(* CODESYS project T1_ARC.project

Project tree, tasks and I/O mapping:
  Device : CODESYS Control Win V3, 3S - Smart Software Solutions GmbH, order no. 305021, version 3.5.7.20
    application Application
      libraries: Standard, * (System); Util, * (System)
      task MainTask (cyclic, interval t#20ms, priority 1) calls PLC_PRG
      program PLC_PRG [FBD]
      global variables GVL_ARC
      Symbols
*)

// Device/Application/GVL_ARC
VAR_GLOBAL
	PV_h: REAL;
	SP_h: REAL;
	KP_h: REAL;
	TN_h: REAL;
	TV_h: REAL;
	u1_MAN: REAL;
	MAN: BOOL;
	RES: BOOL;
	u1_h: REAL;
	PV_K: REAL;
	SP_K: REAL;
	KP_K: REAL;
	TN_K: REAL;
	TV_K: REAL;
	K_MAN: REAL;
	K: REAL;
	PV_f2: REAL;
	SP_f2: REAL;
	KP_f2: REAL;
	TN_f2: REAL;
	TV_f2: REAL;
	f2_MAN: REAL;
	u2: REAL;
	PV_f1: REAL;
END_VAR

// Device/Application/PLC_PRG
PROGRAM PLC_PRG
VAR
	PID_h: PID;
	PID_K: PID;
	PID_f2: PID;
END_VAR

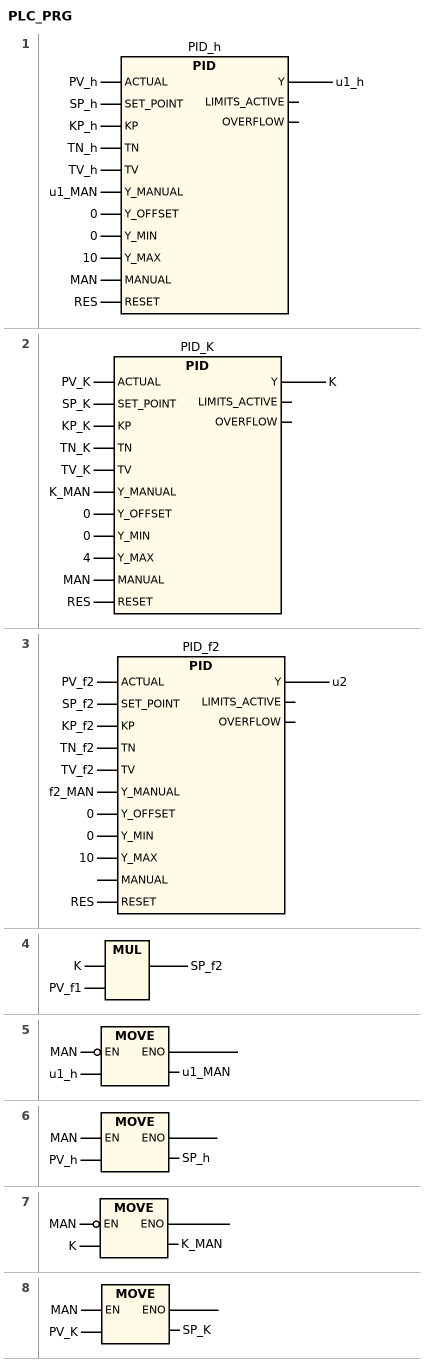
// NETWORK 1
PID_h(
    ACTUAL := PV_h,
    SET_POINT := SP_h,
    KP := KP_h,
    TN := TN_h,
    TV := TV_h,
    Y_MANUAL := u1_MAN,
    Y_OFFSET := 0,
    Y_MIN := 0,
    Y_MAX := 10,
    MANUAL := MAN,
    RESET := RES); // PID
u1_h := PID_h.Y;

// NETWORK 2
PID_K(
    ACTUAL := PV_K,
    SET_POINT := SP_K,
    KP := KP_K,
    TN := TN_K,
    TV := TV_K,
    Y_MANUAL := K_MAN,
    Y_OFFSET := 0,
    Y_MIN := 0,
    Y_MAX := 4,
    MANUAL := MAN,
    RESET := RES); // PID
K := PID_K.Y;

// NETWORK 3
PID_f2(
    ACTUAL := PV_f2,
    SET_POINT := SP_f2,
    KP := KP_f2,
    TN := TN_f2,
    TV := TV_f2,
    Y_MANUAL := f2_MAN,
    Y_OFFSET := 0,
    Y_MIN := 0,
    Y_MAX := 10,
    RESET := RES); // PID
u2 := PID_f2.Y;

// NETWORK 4
SP_f2 := K * PV_f1;

// NETWORK 5
IF NOT MAN THEN u1_MAN := u1_h; END_IF

// NETWORK 6
IF MAN THEN SP_h := PV_h; END_IF

// NETWORK 7
IF NOT MAN THEN K_MAN := K; END_IF

// NETWORK 8
IF MAN THEN SP_K := PV_K; END_IF

END_PROGRAM
